TYPE HugeString : STRING(500000); END_TYPE

(* stored: Version 1.1.0.1, ProductVersion 3.1.4024.12
   DUT HugeString: Id {0b101bb8-f0fa-0a1c-0297-b4645234c57d} *)
